FUNCTION_BLOCK FB_SimulatedIn_DG IMPLEMENTS ITF_Regelschuif_IN_DG

VAR
	internalState : sint;
END_VAR

{warning 'Add method implementation '}
METHOD get : SINT
get := internalState;
END_METHOD

END_FUNCTION_BLOCK

(* stored: Version 1.1.0.1, ProductVersion 3.1.4026.8
   POU FB_SimulatedIn_DG: Id {aac0b935-999d-4985-8292-12706ec9a1c7}, SpecialFunc None
   Method get: Id {79e034de-ecf5-433b-b644-ff4e1cc32dd5} *)
